TYPE DUT_HIM_Probe :
STRUCT
	ActualProbeValue : REAL;
	ActualEncoderValue : REAL;
	Error	: BOOL;
	UpperLimit	: REAL;
	LowerLimit	: REAL;
END_STRUCT
END_TYPE

(* stored: Version 1.1.0.1, ProductVersion 3.1.4024.15
   DUT DUT_HIM_Probe: Id {85d5d163-bb9e-4f0b-9725-b7909fc9c4e0} *)
